FUNCTION_BLOCK Button_HMI
  (* Standard: 61499-2 *)
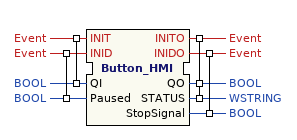
  EVENT_INPUT
    INIT WITH QI;
    INID WITH Paused;
  END_EVENT
  EVENT_OUTPUT
    INITO WITH QO, STATUS;
    INIDO WITH StopSignal;
  END_EVENT
  VAR_INPUT
    QI : BOOL;
    Paused : BOOL;
  END_VAR
  VAR_OUTPUT
    QO : BOOL;
    STATUS : WSTRING;
    StopSignal : BOOL;
  END_VAR
END_FUNCTION_BLOCK
